(* Statuses of the gauges for the switchbox *)
TYPE ST_SBGaugeReadings :
STRUCT
	(* Gauge readings *)
	
	fDPPiraniVal : REAL; // LXLHN:GPI:03
	eDPPiraniState : E_PressureState;
	
	fDPColdCathodeVal : REAL; // LXLHN:GCC:02
	eDPColdCathodeState : E_PressureState;
	
	fPumpStationPirani1Val : REAL; // LXLHN:GPI:01
	ePumpStationPirani1State : E_PressureState;
	
	fPumpStationPirani2Val : REAL; // LXLHN:GPI:02
	ePumpStationPirani2State : E_PressureState;
	
	fPumpStationColdCathodeVal : REAL; // LXLHN:GCC:01
	ePumpStationColdCathodeState : E_PressureState;
END_STRUCT
END_TYPE

(* stored: Version 1.1.0.1, ProductVersion 3.1.4022.18
   DUT ST_SBGaugeReadings: Id {64272b40-03eb-4133-bbf3-046df264c7f8} *)
